// TIA Portal project "teststep" (V17)

(* hardware
DEVICE "S7-1200 station_1"  S7-1200 Station
   slot 0: "Rack_0"  S7-1200 Rack  Rack  V1.0
   slot 1: "PLC_1"  CPU 1214C DC/DC/DC  6ES7 214-1AG40-0XB0  V4.5
*)

// ===== PLC "PLC_1"  CPU 1214C DC/DC/DC =====

VAR_GLOBAL   // PLC tag table "Default tag table"
   "Axes_Y_Pulse" AT %Q0.6 : Bool;
   "Axes_Y_Direction" AT %Q0.7 : Bool;
   "Axes_Y_Pulse(1)" AT %Q0.0 : Bool;
   "Axes_Y_Direction(1)" AT %Q0.1 : Bool;
   "Axes_X_Pulse" AT %Q0.4 : Bool;
   "Axes_X_Direction" AT %Q0.5 : Bool;
   "Axes_X_Pulse(1)" AT %Q0.2 : Bool;
   "Axes_X_Direction(1)" AT %Q0.3 : Bool;
   "Tag_1" AT %I0.1 : Bool;
   "Tag_2" AT %Q1.0 : Bool;
   "Tag_3" AT %M1.0 : Bool;
   "Axes_X_LowHwLimitSwitch" AT %I0.0 : Bool;
END_VAR

DATA_BLOCK "Axes_X"   // DB1, Motion_DB
{ S7_Optimized_Access := 'TRUE' }
AUTHOR : SIMATIC
FAMILY : BasicMC
NAME : TO_PosAx
VERSION : 8.0
// stored: InstanceOfName TO_PositioningAxis
"TO_PositioningAxis"
BEGIN
   // Axis.PositionLimitsMax_AddressCU = %I0.0
   // Axis.PositionLimitsMin_AddressCU = %I0.1
   // Axis.HomingReferencePointSwitch_AddressCU = %I0.1
   // Axis.DirectionOutputEnabledCU = TRUE
   // Axis.OnlinePtoIndexCU = 1
   // Axis.OnlinePtoModeCU = 16#0000_0002
   // Axis.SelectedChannel2EnumCU = %Q0.3
   // Axis.SelectedChannel1EnumCU = %Q0.2
   // Pulse.MinDeltaDeltaFrequencyCU = 0.004
   // Pulse.MaxDeltaDeltaFrequencyCU = 1.0E+10
   // Pulse.MinDeltaFrequencyCU = 0.005
   // Pulse.MaxDeltaFrequencyCU = 9.5E+9
   // Pulse.MinFrequencyCU = 1.0
   // Pulse.MaxFrequencyCU = 100000.0
   // Pulse.OutputSourceCU = 16#0000_0000
   // Axis.SelectPTO = 1
   // Axis.LengthUnit.LastDistance = -1
END_DATA_BLOCK

ORGANIZATION_BLOCK "Main"   // OB1, LAD, ProgramCycle
TITLE = "Main Program Sweep (Cycle)"
{ S7_Optimized_Access := 'TRUE' }
VERSION : 0.1
   VAR_INPUT
      Initial_Call : Bool;   // Initial call of this OB
      Remanence : Bool;   // =True, if remanent data are available
   END_VAR
BEGIN
END_ORGANIZATION_BLOCK